FUNCTION_BLOCK FINAL Action_I_Observer_

METHOD Perform
VAR_INPUT
    applyCaseNumber : INT;
END_VAR
VAR_IN_OUT
	item : I_Observer;
END_VAR
CASE applyCaseNumber OF
    1 :
    item.OnUpdate();
    2 :
    item.OnError();
ELSE
    RETURN;
END_CASE
END_METHOD

END_FUNCTION_BLOCK

(* stored: Version 1.1.0.1, ProductVersion 3.1.4024.6
   POU Action_I_Observer_: Id {8a2bf32b-de93-4ece-9af4-43f93abc4c97}, SpecialFunc None
   Method Perform: Id {01b2032b-41a7-42a3-8c6a-d654fad2b1f1} *)
